TYPE Axis_OUTPUT :
STRUCT
	Control_Word AT%Q*:WORD;
	Target_Position AT%Q*:DINT;
	Profile_Velocity AT%Q*:UDINT;
	Max_Velocity AT%Q*:UDINT;
	Mode_of_Operation AT%Q* :BYTE:=1;
	Target_Torque AT%Q* :INT:=0;
	Max_Torque AT%Q*: UINT :=0;
END_STRUCT
END_TYPE

(* stored: Version 1.1.0.1, ProductVersion 3.1.4024.12
   DUT Axis_OUTPUT: Id {97f69d60-d002-4272-bb59-28e812e064b0} *)
